FUNCTION "LKinCtrl_InitTODataStore" : "LKinCtrl_typePnPInitTOData"
TITLE = LKinCtrl_InitTODataStore
{ S7_Optimized_Access := 'TRUE' }
AUTHOR : 'handling.team.automation@siemens.com'
FAMILY : LKinCtrl
VERSION : 5.0
//Store specific TO data
   VAR_IN_OUT
      axesGroup {InstructionName := 'TO_Kinematics'; LibVersion := '9.0'} : TO_Kinematics;   // Reference to axes group
   END_VAR


BEGIN
	//=============================================================================
	// SIEMENS AG
	// (c)Copyright 2023
	//-----------------------------------------------------------------------------
	// Library:       LKinCtrl
	// Tested with:   S7-1518TF-4 PN/DP, FW V3.1
	// Engineering:   TIA Portal V19
	// Restrictions:  ---
	// Requirements:  S7-1500T, FW V3.0
	// Functionality: Store specific TO data
	// Support: tech.team.motioncontrol@siemens.com
	// Note: Parameter comments are only available in language 'English (United States)'
	//-----------------------------------------------------------------------------
	// Change log table:
	// Version  Date       Expert in charge Changes applied
	// 01.00.00 21.09.2023 SF               First released version
	//=============================================================================

	//Blending length factor
	#LKinCtrl_InitTODataStore.factorBlendingLength := #axesGroup.Transition.FactorBlendingLength;
	//Orientation dynamics
	#LKinCtrl_InitTODataStore.orientationDefaults.velocity := #axesGroup.DynamicDefaults.Orientation.Velocity;
	#LKinCtrl_InitTODataStore.orientationDefaults.acceleration := #axesGroup.DynamicDefaults.Orientation.Acceleration;
	#LKinCtrl_InitTODataStore.orientationDefaults.deceleration := #axesGroup.DynamicDefaults.Orientation.Deceleration;
	#LKinCtrl_InitTODataStore.orientationDefaults.jerk := #axesGroup.DynamicDefaults.Orientation.Jerk;
END_FUNCTION

